PROGRAM MeinProgramm
VAR
	T1: ton;
	T2: ton;
END_VAR

T1(IN:=NOT t2.Q, pt:=T#1S);
T2(in:=t1.Q,pt:=T#1S);

DaDi.P1:= T1.Q;

END_PROGRAM

(* stored: Version 1.1.0.1, ProductVersion 3.1.4024.5
   POU MeinProgramm: Id {35e6b61e-d309-4819-ad74-2516ed18df2b}, SpecialFunc None *)
